FUNCTION_BLOCK PUBLIC FB_ItalianPizzaMargherita EXTENDS FB_PizzaItalianStyle
VAR_INPUT
END_VAR
VAR_OUTPUT
END_VAR
VAR
	bCheese		: BOOL := TRUE;
	bTomato		: BOOL := TRUE;
END_VAR

PROPERTY PUBLIC bHasCheese : BOOL
GET
bHasCheese := this^.bCheese;
END_GET
SET
this^.bCheese := bHasCheese;
END_SET
END_PROPERTY

PROPERTY PUBLIC bHasTomato : BOOL
GET
bHasTomato := this^.bTomato;
END_GET
SET
this^.bTomato := bHasTomato;
END_SET
END_PROPERTY

METHOD PUBLIC GetPrice : LREAL
GetPrice := SUPER^.GetPrice();
IF (THIS^.bCheese) THEN
	GetPrice := GetPrice + 1.1;
END_IF
IF (THIS^.bTomato) THEN
	GetPrice := GetPrice + 0.9;
END_IF
END_METHOD

END_FUNCTION_BLOCK

(* stored: Version 1.1.0.1, ProductVersion 3.1.4022.12
   POU FB_ItalianPizzaMargherita: Id {01b9f8de-cd87-4aca-aa43-d6d501bcb44f}, SpecialFunc None
   Property bHasCheese: Id {a2b0bc13-3c5a-4d6c-a81a-3623047e5056}
   Get Get: Id {4f303c06-fd8d-4486-8713-57c2f4ed2563}
   Set Set: Id {d6b4790b-dca6-43a2-9046-8771cdc5ba31}
   Property bHasTomato: Id {f05c209a-a7ca-473e-9b0c-1d314637b511}
   Get Get: Id {6650a8d4-7df9-4081-8ea2-245fd3bdab9f}
   Set Set: Id {2c78b884-ea64-4165-90f4-cd76947a5fee}
   Method GetPrice: Id {16fe620a-7ddf-4849-ad7e-214e84293023} *)
